{attribute 'qualified_only'}
{attribute 'strict'}
{attribute 'to_string'}
// 料盘流程错误码。
// 保留原范围，并定义本次异常保护错误码：16#6200～16#62FF。
TYPE E_TrayErrorCode :
(
    None         := 16#0000,
    ReservedBase := 16#6200,
    MotionCommandRejected := 16#6211,
    MotionCommandAborted  := 16#6212,
    MotionTimeout         := 16#6213,
    PlannedTrayMissing    := 16#6214, // 计划层真正入架取盘前稳定缺盘
    ReservedEnd  := 16#62FF
) UDINT;
END_TYPE

(* stored: Version 1.1.0.1, ProductVersion 3.1.4026.20
   DUT E_TrayErrorCode: Id {03683152-6a0b-4c7f-986c-0e6b9ba04ab6} *)
